FUNCTION_BLOCK ConveyorCtrl (* Template for an empty basic function block *)
  (* Standard: 61499-2 *)
  (* Version 1.0, 2018-09-13, az *)
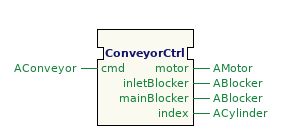
  SOCKETS
    cmd : AConveyor;
  END_SOCKETS
  PLUGS
    motor : AMotor;
    inletBlocker : ABlocker;
    mainBlocker : ABlocker;
    index : ACylinder;
  END_PLUGS
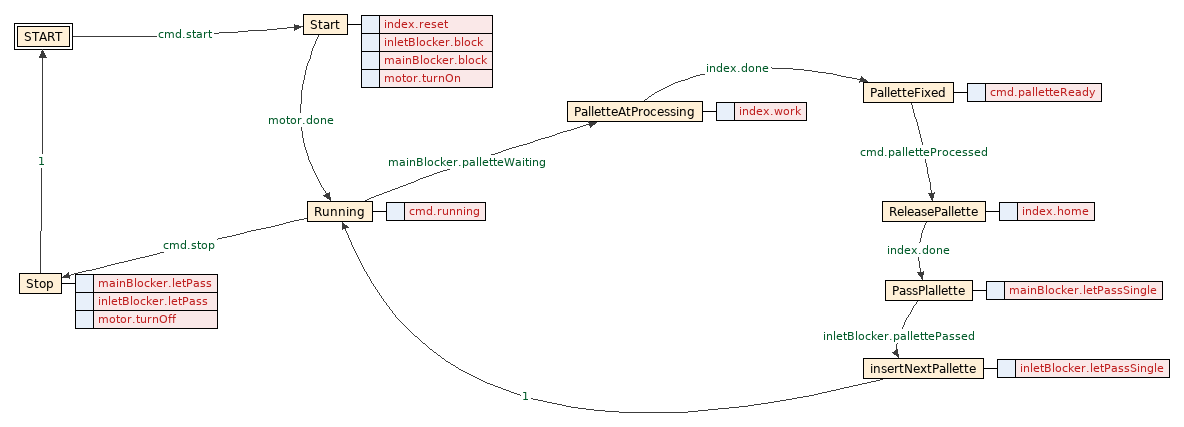
  EC_STATES
    START; (* Initial State *)
    Start : -> index.reset, -> inletBlocker.block, -> mainBlocker.block, -> motor.turnOn;
    Running : -> cmd.running;
    PalletteAtProcessing : -> index.work;
    PalletteFixed : -> cmd.palletteReady;
    ReleasePallette : -> index.home;
    PassPlallette : -> mainBlocker.letPassSingle;
    insertNextPallette : -> inletBlocker.letPassSingle;
    Stop : -> mainBlocker.letPass, -> inletBlocker.letPass, -> motor.turnOff;
  END_STATES
  EC_TRANSITIONS
    START TO Start := cmd.start;
    Start TO Running := motor.done;
    Running TO PalletteAtProcessing := mainBlocker.palletteWaiting;
    PalletteAtProcessing TO PalletteFixed := index.done;
    PalletteFixed TO ReleasePallette := cmd.palletteProcessed;
    ReleasePallette TO PassPlallette := index.done;
    PassPlallette TO insertNextPallette := inletBlocker.pallettePassed;
    insertNextPallette TO Running := 1;
    Running TO Stop := cmd.stop;
    Stop TO START := 1;
  END_TRANSITIONS
END_FUNCTION_BLOCK
